(*In development phase*)
FUNCTION_BLOCK FB_ModbusMasterTcpIp
VAR
	sName			:		STRING;
	iScantime		:		UINT := 50;
	iTimeout		:		UINT := 1000;//1000ms
	iErrorID		:		UDINT;
	bBusy			: 		BOOL;
	bError			:		BOOL;
	iStepGeneral	: 		E_ModBusMasterState;
	iStepRunning	:		E_ModbusMasterStateRun;
	bFirstCycle		:		BOOL;
	bRun			:		BOOL;
	bStop			: 		BOOL;

	FbMBReadCoils	: 		FB_MBReadCoils;
	FbMBReadInputs  : 		FB_MBReadInputs;
	FbMBReadRegs	:		FB_MBReadRegs;
	FbMBReadInputRegs	: 	FB_MBReadInputRegs;
	FbWriteSingleCoil 	:	FB_MBWriteSingleCoil;
	FbMBWriteSingleReg	:	FB_MBWriteSingleReg;
	FbMBWriteCoils		: 	FB_MBWriteCoils;
	FbMBWriteRegs		:	FB_MBWriteRegs;
	ipModbusSlave	:		ARRAY [1..247] OF I_ModbusSlaveTcp;
	iAmountSlave	: 		UINT;
	
	iLoopSlave		:		UINT	:= 1;
	iLoopAdr		:		UINT;
	iQuantity 		: 		POINTER TO WORD;
	iMBAddr 		: 		POINTER TO WORD;
    arrData			: 		ARRAY [0..255] OF WORD;
	
	sIPAddr			: STRING(15);
	nTCPPort		: UINT;
	UnitId			: BYTE;
	Quantity		: WORD;
	MBAddr			: WORD;
	cbLength 		: UINT;
	pMemoryAddr		: POINTER TO BYTE;
	pDataWrite		: POINTER TO WORD;

	bexecute		: BOOL;
	
	tCalculateTimeRW	: TON;
	tTimerScanDelay		: TON;
	nNumberFaultRW		: UINT;
	eModbusFunction		: E_ModbusFunction;
	peModbusFunction 	: POINTER TO WORD;
END_VAR

StateMachine();
bRun := iStepGeneral=E_ModBusMasterState.Running ;
bStop := iStepGeneral=E_ModBusMasterState.Stop;

PROPERTY AnyError : BOOL
GET
AnyError 	:= bError;
END_GET
END_PROPERTY

PROPERTY Busy : BOOL
GET
Busy := bBusy;
END_GET
END_PROPERTY

PROPERTY CycleTimeMeasure : Time
GET
CycleTimeMeasure := tCalculateTimeRW.ET;
END_GET
END_PROPERTY

PROPERTY ErrorID : UDINT;
GET
ErrorID := iErrorID;
END_GET
END_PROPERTY

PROPERTY Name : STRING
GET
Name := sName;
END_GET
SET
sName := Name;
END_SET
END_PROPERTY

PROPERTY ReadData : ARRAY [0..255] OF Word
GET
ReadData := arrData;
END_GET
END_PROPERTY

PROPERTY ReadDataSize : uint
GET
ReadDataSize := INT_TO_UINT(SIZEOF(arrData));
END_GET
END_PROPERTY

METHOD RegisterSlave : BOOL
VAR_INPUT
	ModbusSlave		:		I_ModbusSlaveTcp;
END_VAR
VAR
	iLoop	:	UINT;
	bExists	:	BOOL;
END_VAR
FOR iLoop := 1 TO iAmountSlave DO
	IF ipModbusSlave[iLoop] = ModbusSlave THEN
		bExists := TRUE;
		iLoop := iAmountSlave;// end loop for command
	END_IF
END_FOR 
IF NOT bExists THEN
	iAmountSlave := iAmountSlave + 1;
	ipModbusSlave[iAmountSlave] := ModbusSlave;
END_IF
END_METHOD

METHOD Reset : BOOL
bError := FALSE;
iErrorID := 0;
bError := FALSE;
iStepGeneral := E_ModBusMasterState.Stop;
iStepRunning := E_ModbusMasterStateRun.CheckNumberSlaveRegistered;
iLoopSlave := 1;
iLoopAdr := 0;
FbMBReadCoils(bExecute := FALSE);
FbMBReadInputs(bExecute := FALSE);
FbMBReadRegs(bExecute := FALSE);
FbMBReadInputRegs(bExecute := FALSE);
FbWriteSingleCoil(bExecute := FALSE);
FbMBWriteSingleReg(bExecute := FALSE);
FbMBWriteCoils(bExecute := FALSE);
FbMBWriteRegs(bExecute := FALSE);
Reset := TRUE;
END_METHOD

METHOD Run : BOOL /// call from FB_modbus
iStepGeneral := E_ModBusMasterState.Running;
bRun := TRUE;
Run := TRUE;
END_METHOD

PROPERTY ScanTime : UINT
GET
ScanTime := iScantime;
END_GET
SET
iScantime := ScanTime;
END_SET
END_PROPERTY

METHOD protected StateMachine : BOOL (*State machine of unit*)
CASE iStepGeneral OF
		E_ModBusMasterState.Running: 
			StateRunning();
						
		E_ModBusMasterState.stop:
			StateStopping();
END_CASE
END_METHOD

METHOD PROTECTED StateRunning : BOOL (* Unit is uninitialized*)
VAR 
	

	
END_VAR
CASE iStepRunning OF
	E_ModbusMasterStateRun.CheckNumberSlaveRegistered: // Trigger
		tCalculateTimeRW(
			IN := TRUE,
			PT := T#5M
		);	
		IF iAmountSlave > 0 THEN
			iStepRunning := E_ModbusMasterStateRun.SetParametersRead;
		END_IF
			
	E_ModbusMasterStateRun.SetParametersRead: // Set parameters
		IF ipModbusSlave[iLoopSlave].NumAddRegionRead <> 0 
			AND iLoopAdr <= (ipModbusSlave[iLoopSlave].NumAddRegionRead - 1) 
		THEN
			sIPAddr := ipModbusSlave[iLoopSlave].IpAddr;
			nTCPPort := ipModbusSlave[iLoopSlave].TcpPort;
			iQuantity := ipModbusSlave[iLoopSlave].AddressRead + ((iLoopAdr * 3 + 1) * SIZEOF(WORD));// arrAddressRead[iloopAdr][1] in Slave
			iMBAddr := ipModbusSlave[iLoopSlave].AddressRead + ((iLoopAdr * 3) * SIZEOF(WORD));// arrAddressRead[iloopAdr][0] in Slave
			UnitID := ipModbusSlave[iLoopSlave].UnitID;
			Quantity :=	iQuantity^;
			MBAddr := iMBAddr^;
			cbLength := SIZEOF(arrData);
			pMemoryAddr	:= ADR(arrData);
			peModbusFunction := ipModbusSlave[iLoopSlave].AddressRead + ((iLoopAdr * 3 + 2) * SIZEOF(WORD)); // arrAddressRead[iloopAdr][2] in Slave
			eModbusFunction := peModbusFunction^;
			iStepRunning := E_ModbusMasterStateRun.SendRequestRead;
		ELSE 
			iLoopAdr := 0;
			iStepRunning := E_ModbusMasterStateRun.ReturnReadDone;
		END_IF

			
	E_ModbusMasterStateRun.SendRequestRead: // Send request
		CASE eModbusFunction OF
			E_ModbusFunction.ReadHoldingRegisters:
				FbMBReadRegs(
					sIPAddr := sIPAddr,
					nTCPPort := nTCPPort,
					nUnitID := UnitID,
					nQuantity := Quantity,
					nMBAddr := MBAddr,
					cbLength := cbLength,
					pDestAddr := pMemoryAddr,
					bExecute := TRUE,
					tTimeout := UINT_TO_TIME(iTimeout),
					bBusy => bBusy,
					bError => bError,
					nErrId => iErrorId,
				);
			
			E_ModbusFunction.ReadInputRegisters:
				FbMBReadInputRegs(
					sIPAddr := sIPAddr,
					nTCPPort := nTCPPort,
					nUnitID := UnitID,
					nQuantity := Quantity,
					nMBAddr := MBAddr,
					cbLength := cbLength,
					pDestAddr := pMemoryAddr,
					bExecute := TRUE,
					tTimeout := UINT_TO_TIME(iTimeout),
					bBusy => bBusy,
					bError => bError,
					nErrId => iErrorId,
				);
			
		END_CASE
		iStepRunning := E_ModbusMasterStateRun.WaitReadRespond;
						
	E_ModbusMasterStateRun.WaitReadRespond:
		FbMBReadRegs(bExecute := FALSE);
		FbMBReadInputRegs(bExecute := FALSE);
		IF NOT bBusy AND NOT bError THEN
			ipModbusSlave[iLoopSlave].ModbusErrorID := iErrorID;
			iStepRunning := E_ModbusMasterStateRun.ConvertRawData;
			nNumberFaultRW := 0;
		END_IF
		
		IF bError AND NOT bBusy THEN
			ipModbusSlave[iLoopSlave].ModbusErrorID := iErrorID;
			iStepRunning := E_ModbusMasterStateRun.ReturnReadDone;
		END_IF
	
	E_ModbusMasterStateRun.ConvertRawData: 
		ipModbusSlave[iLoopSlave].Convert(
			iRegionNo := iLoopAdr,
		 	pReadData := ADR(arrData)
		);
		iLoopAdr := iLoopAdr + 1;
		iStepRunning := E_ModbusMasterStateRun.CheckNumberSlaveRegistered;

	E_ModbusMasterStateRun.ReturnReadDone: // Return, done
		iStepRunning := E_ModbusMasterStateRun.SetParametersWrite;
		iLoopAdr := 0;

	E_ModbusMasterStateRun.SetParametersWrite :
		IF  ipModbusSlave[iLoopSlave].NumAddRegionWrite <> 0
		AND iLoopAdr <= ipModbusSlave[iLoopSlave].NumAddRegionWrite - 1 
		THEN // iLoopAdr start from 1
			sIPAddr := ipModbusSlave[iLoopSlave].IpAddr;
			nTCPPort := ipModbusSlave[iLoopSlave].TcpPort;
			iMBAddr := ipModbusSlave[iLoopSlave].AddressWrite + (iLoopAdr * 11 * SIZEOF(WORD));// return address word contain value address( modbus) 
			pDataWrite := ipModbusSlave[iLoopSlave].AddressWrite + ((iLoopAdr * 11 + 2) * SIZEOF(WORD));
			iQuantity := ipModbusSlave[iLoopSlave].AddressWrite + ((iLoopAdr * 11 + 1) * SIZEOF(WORD));
			peModbusFunction := ipModbusSlave[iLoopSlave].AddressWrite + ((iLoopAdr * 11 + 10) * SIZEOF(WORD));
			eModbusFunction := peModbusFunction^;
			UnitID 	:=		ipModbusSlave[iLoopSlave].UnitID;
			Quantity	:=	iQuantity^;
			MBAddr	:=		iMBAddr^;
			cbLength	:= 	Quantity * 2;
			pMemoryAddr	:= 	pDataWrite;
			iStepRunning := E_ModbusMasterStateRun.SendRequestWrite;
		ELSE 
			iStepRunning := E_ModbusMasterStateRun.ReturnWriteDone;
		END_IF

	E_ModbusMasterStateRun.SendRequestWrite :
		CASE eModbusFunction OF
			E_ModbusFunction.WriteMultipleCoils:
				FbMBWriteCoils(
					sIPAddr := sIPAddr,
					nTCPPort := nTCPPort,
					nUnitID := UnitID,
					nQuantity := Quantity,
					nMBAddr := MBAddr,
					cbLength := cbLength,
					pSrcAddr := pMemoryAddr,
					bExecute := TRUE,
					tTimeout := UINT_TO_TIME(iTimeout),
					bBusy => bBusy,
					bError => bError,
					nErrId => iErrorId,
				);
													
			E_ModbusFunction.WriteMultipleRegisters:
				FbMBWriteRegs(
					sIPAddr := sIPAddr,
					nTCPPort := nTCPPort,
					nUnitID := UnitID,
					nQuantity := Quantity,
					nMBAddr := MBAddr,
					cbLength := cbLength,
					pSrcAddr := pMemoryAddr,
					bExecute := TRUE,
					tTimeout := UINT_TO_TIME(iTimeout),
					bBusy => bBusy,
					bError => bError,
					nErrId => iErrorId,
				);
											
			E_ModbusFunction.WriteSingleCoil:
				FbWriteSingleCoil(
					sIPAddr := sIPAddr,
					nTCPPort := nTCPPort,
					nUnitID := UnitID,
					nMBAddr := MBAddr,
					nValue := pDataWrite^,
					bExecute := TRUE,
					tTimeout := UINT_TO_TIME(iTimeout),
					bBusy => bBusy,
					bError => bError,
					nErrId => iErrorId,
				);
			E_ModbusFunction.WriteSingleRegister:
				FbMBWriteSingleReg(
					sIPAddr := sIPAddr,
					nTCPPort := nTCPPort,
					nUnitID := UnitID,
					nMBAddr := MBAddr,
					nValue := pDataWrite^,
					bExecute := TRUE,
					tTimeout := UINT_TO_TIME(iTimeout),
					bBusy => bBusy,
					bError => bError,
					nErrId => iErrorId,
				);
		END_CASE
		
		iStepRunning := E_ModbusMasterStateRun.WaitWriteRespond;
	
	E_ModbusMasterStateRun.WaitWriteRespond :
		FbMBWriteCoils(bExecute := FALSE);
		FbMBWriteRegs(bExecute := FALSE);
		FbWriteSingleCoil(bExecute := FALSE);	
		FbMBWriteSingleReg(bExecute := FALSE);
		IF NOT bBusy AND NOT bError THEN
			ipModbusSlave[iLoopSlave].ModbusErrorID := iErrorID;
			iStepRunning := E_ModbusMasterStateRun.SetParametersWrite;
			nNumberFaultRW := 0;
			iLoopAdr := iLoopAdr + 1;
		END_IF
		IF bError AND NOT bBusy THEN
			ipModbusSlave[iLoopSlave].ModbusErrorID := iErrorID;
			iStepRunning := E_ModbusMasterStateRun.ReturnWriteDone ;
		END_IF
	
	 E_ModbusMasterStateRun.ReturnWriteDone :
		iLoopAdr := 0;
		iLoopSlave := iLoopSlave + 1;// next slave
		IF iLoopSlave > iAmountSlave THEN
			iLoopSlave := 1;
		END_IF
		tTimerScanDelay( 
			IN := TRUE,
			PT := UINT_TO_TIME(iScantime)
		);
		IF tTimerScanDelay.Q THEN
			tTimerScanDelay( IN := FALSE);
			tCalculateTimeRW(in := FALSE);
		 	iStepRunning := E_ModbusMasterStateRun.CheckNumberSlaveRegistered;
		END_IF
			
END_CASE
END_METHOD

METHOD protected StateStopping : BOOL (* Unit is uninitialized*)
iStepRunning	:= E_ModbusMasterStateRun.CheckNumberSlaveRegistered;
iLoopSlave		:= 1;
iLoopAdr		:= 0;
FbMBReadCoils(bExecute := FALSE);
FbMBReadInputs(bExecute := FALSE);
FbMBReadRegs(bExecute := FALSE);
FbMBReadInputRegs(bExecute := FALSE);
FbWriteSingleCoil(bExecute := FALSE);
FbMBWriteSingleReg(bExecute := FALSE);
FbMBWriteCoils(bExecute := FALSE);
FbMBWriteRegs(bExecute := FALSE);
END_METHOD

METHOD Stop : BOOL
iStepGeneral := E_ModBusMasterState.stop;
bStop := TRUE;
Stop := TRUE;
END_METHOD

PROPERTY Stopped : bool
GET
Stopped := bStop;
END_GET
END_PROPERTY

PROPERTY Timeout : UINT // in milisecond, if not respond in this time , error will raise
GET
Timeout := iTimeout;
END_GET
SET
iTimeout := Timeout;
END_SET
END_PROPERTY

END_FUNCTION_BLOCK

(* stored: Version 1.1.0.1, ProductVersion 3.1.4024.12
   POU FB_ModbusMasterTcpIp: Id {98074c56-eb83-4935-8b15-ba49c7be4882}, SpecialFunc None
   Folder Methods: Id {41e40c12-4e9c-40cd-af28-94fcec93fe43}
   Folder Property: Id {834abddb-6368-4df6-8748-8fa11929b403}
   Folder StateMachine: Id {16c36b51-8505-4e5a-8071-b60bab127d37}
   Property AnyError: Id {a4612b41-7055-4a62-9846-e1fb76272b9e}
   Get Get: Id {12b3606a-c594-409a-be94-422716f0d01c}
   Property Busy: Id {95302009-422e-4d1d-8f8f-2d6e8be28375}
   Get Get: Id {49de5639-bb4c-475f-8f18-de4e11b5d305}
   Property CycleTimeMeasure: Id {93728dd0-ab6c-483f-822b-e4e8226a06a2}
   Get Get: Id {96700f1c-8d25-48c1-90f0-1397a9b8898f}
   Property ErrorID: Id {f3d8ab52-f5eb-42af-b956-c85767f4af04}
   Get Get: Id {b89fb2c4-5541-4c73-8b9f-0e243678462f}
   Property Name: Id {95628104-8e0e-4c95-86ba-017d5c440d47}
   Get Get: Id {4b1de093-e9e9-4503-bb4a-5198ed798a1e}
   Set Set: Id {64c7ad31-5de6-4152-81bb-37a6dd6b6d64}
   Property ReadData: Id {ab9353cd-951c-4dec-860b-3a19747bf71d}
   Get Get: Id {4075d516-90aa-47fa-9607-9ffe7d25021f}
   Property ReadDataSize: Id {d6bac55e-904c-48d7-b040-b191eb8eeaac}
   Get Get: Id {ed49f154-d511-4a0b-9e67-e95fcf97a33c}
   Method RegisterSlave: Id {3e82ec34-bcea-40ad-bfd3-3c4a6c79618c}
   Method Reset: Id {2bbe55ae-94a3-4e44-ba94-163ab9032719}
   Method Run: Id {b0399b31-e9e7-4a38-97a6-d96564f950bd}
   Property ScanTime: Id {02f8582d-dd7c-49a8-8e86-3cb1ed7fee5c}
   Get Get: Id {ea98ff6b-5e39-46d3-a604-3a4a5d1add54}
   Set Set: Id {02190077-5ae3-4f78-b4b5-61732a283290}
   Method StateMachine: Id {17fac4bf-ff20-4332-8f26-ee2610e0eb8a}
   Method StateRunning: Id {14f3e285-b5fe-4b2d-a981-fbf097c16e04}
   Method StateStopping: Id {28c96804-c7c0-49fe-aec4-36f59f92fb28}
   Method Stop: Id {29c55c48-0ff2-4962-8292-2c50edc10688}
   Property Stopped: Id {15683197-244e-4d5b-a3a9-ede92924424b}
   Get Get: Id {ecb3b88b-647c-4986-a19b-e660939b3957}
   Property Timeout: Id {796dcbbb-13e6-41c3-944b-11e87005ee64}
   Get Get: Id {b91dca54-f5c4-496f-9110-ea5fe355241f}
   Set Set: Id {449789ce-70a7-4b9d-b930-d8d570fb1c19} *)
